// TIA Portal V18 export
FUNCTION "Proxy_General" : Void   // FC59000, LAD
{ S7_Optimized_Access := 'TRUE' }
VERSION : 0.1
// stored: AutoNumber false, IsIECCheckEnabled false, SetENOAutomatically false, UDAEnableTagReadback false
BEGIN

REGION Network 1
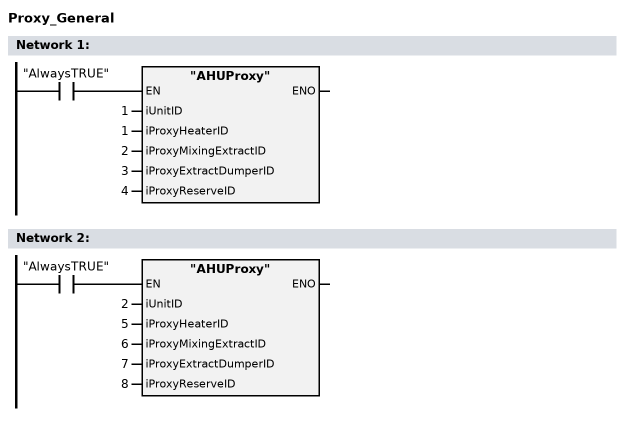
   RUNG wire#powerrail
      Contact( "AlwaysTRUE" )
      "AHUProxy"(iUnitID := 1, iProxyHeaterID := 1, iProxyMixingExtractID := 2, iProxyExtractDumperID := 3, iProxyReserveID := 4)
   END_RUNG
   // the same network as SCL:
   IF "AlwaysTRUE" THEN
       "AHUProxy"(iUnitID := 1,
                  iProxyHeaterID := 1,
                  iProxyMixingExtractID := 2,
                  iProxyExtractDumperID := 3,
                  iProxyReserveID := 4);
   END_IF;
END_REGION

REGION Network 2
   RUNG wire#powerrail
      Contact( "AlwaysTRUE" )
      "AHUProxy"(iUnitID := 2, iProxyHeaterID := 5, iProxyMixingExtractID := 6, iProxyExtractDumperID := 7, iProxyReserveID := 8)
   END_RUNG
   // the same network as SCL:
   IF "AlwaysTRUE" THEN
       "AHUProxy"(iUnitID := 2,
                  iProxyHeaterID := 5,
                  iProxyMixingExtractID := 6,
                  iProxyExtractDumperID := 7,
                  iProxyReserveID := 8);
   END_IF;
END_REGION
END_FUNCTION
